// TIA Portal V17 export
// export: Created 2024-01-30T08:49:17.2969584Z, ExportSetting WithDefaults, DisplayName Totally Integrated Automation Portal, DisplayVersion V17 Update 6, DisplayName TIA Portal Openness, DisplayVersion V17 Update 6, DisplayName TIA Portal Version Control Interface, DisplayVersion V17, DisplayName STEP 7 Professional, DisplayVersion V17 Update 6, DisplayName STEP 7 Safety, DisplayVersion V17 Update 6, DisplayName WinCC Advanced, DisplayVersion V17 Update 6
TYPE "UDT_FESTO_CMMT_IN"
// stored: IsFailsafeCompliant false
   STRUCT
      ModePos : Int;
      EnableAxis : Bool;
      CancelTraversing : Bool;
      IntermediateStop : Bool;
      Positive : Bool;
      Negative : Bool;
      Jog1 : Bool;
      Jog2 : Bool;
      FlyRef : Bool;
      AckError : Bool;
      ExecuteMode : Bool;
      ReleaseBrake : Bool;
      TraveltoFixStop : Bool;
      Position : DInt;
      Velocity : DInt;
      OverV : Int := 100;
      OverAcc : Int := 100;
      OverDec : Int := 100;
      ConfigEPos : DWord := 16#0000_0007;
      BaseSpeedValue : Real;
      HWIDSTW : HW_IO;
      HWIDZSW : HW_IO;
   END_STRUCT;
END_TYPE
